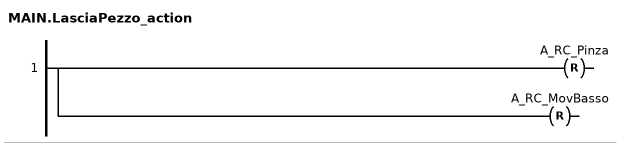
[picture p96: MAIN.LasciaPezzo_action (LD)]
_LD_ (* Ladder Diagram *)
NETWORK 1
	* --- (R A_RC_Pinza) (R A_RC_MovBasso)
_END_LD_
(* the same logic as Structured Text *)
(* Network 1 *)
A_RC_Pinza := FALSE;
A_RC_MovBasso := FALSE;
END_ACTION

ACTION PinzaSet21_action:
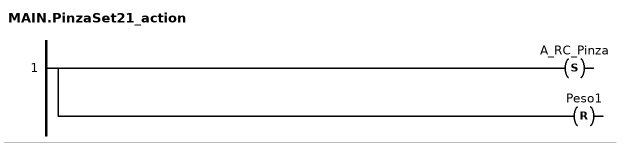
_LD_ (* Ladder Diagram *)
NETWORK 1
	* --- (S A_RC_Pinza) (R Peso1)
_END_LD_
(* the same logic as Structured Text *)
(* Network 1 *)
A_RC_Pinza := TRUE;
Peso1 := FALSE;
END_ACTION

ACTION MovA1_action:
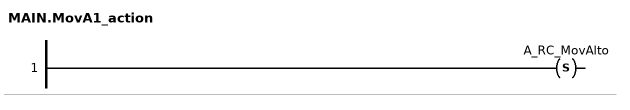
_LD_ (* Ladder Diagram *)
NETWORK 1
	* --- (S A_RC_MovAlto)
_END_LD_
(* the same logic as Structured Text *)
(* Network 1 *)
A_RC_MovAlto := TRUE;
END_ACTION

ACTION MovS1RA_action:
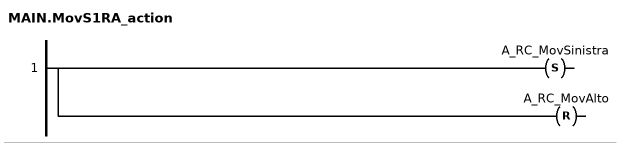
_LD_ (* Ladder Diagram *)
NETWORK 1
	* --- (S A_RC_MovSinistra) (R A_RC_MovAlto)
_END_LD_
(* the same logic as Structured Text *)
(* Network 1 *)
A_RC_MovSinistra := TRUE;
A_RC_MovAlto := FALSE;
END_ACTION

ACTION PinzaSet22_action:
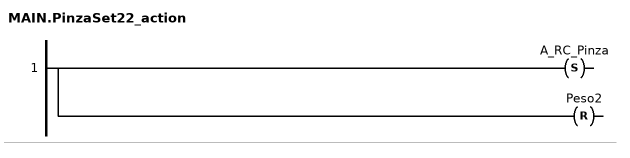
_LD_ (* Ladder Diagram *)
NETWORK 1
	* --- (S A_RC_Pinza) (R Peso2)
_END_LD_
(* the same logic as Structured Text *)
(* Network 1 *)
A_RC_Pinza := TRUE;
Peso2 := FALSE;
END_ACTION

ACTION MovA2_action:
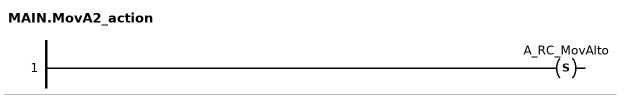
_LD_ (* Ladder Diagram *)
NETWORK 1
	* --- (S A_RC_MovAlto)
_END_LD_
(* the same logic as Structured Text *)
(* Network 1 *)
A_RC_MovAlto := TRUE;
END_ACTION

ACTION MovS2RA_action:
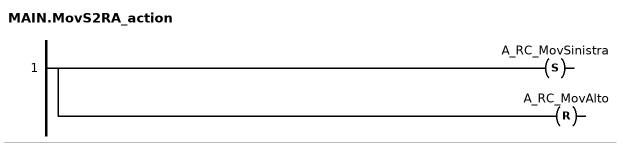
_LD_ (* Ladder Diagram *)
NETWORK 1
	* --- (S A_RC_MovSinistra) (R A_RC_MovAlto)
_END_LD_
(* the same logic as Structured Text *)
(* Network 1 *)
A_RC_MovSinistra := TRUE;
A_RC_MovAlto := FALSE;
END_ACTION

ACTION PinzaSet23_action:
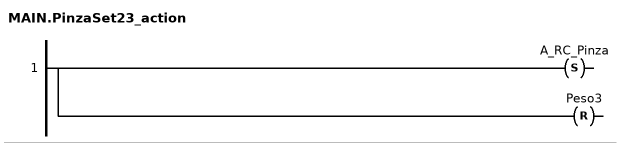
_LD_ (* Ladder Diagram *)
NETWORK 1
	* --- (S A_RC_Pinza) (R Peso3)
_END_LD_
(* the same logic as Structured Text *)
(* Network 1 *)
A_RC_Pinza := TRUE;
Peso3 := FALSE;
END_ACTION

ACTION MovA3_action:
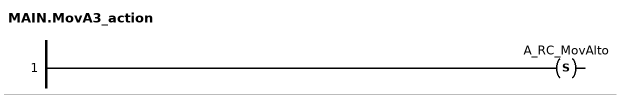
_LD_ (* Ladder Diagram *)
NETWORK 1
	* --- (S A_RC_MovAlto)
_END_LD_
(* the same logic as Structured Text *)
(* Network 1 *)
A_RC_MovAlto := TRUE;
END_ACTION

ACTION MovS3RA_action:
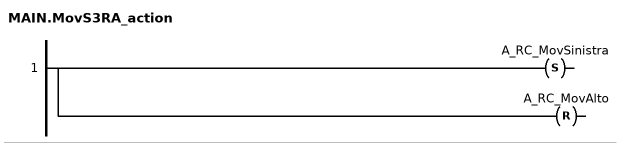
_LD_ (* Ladder Diagram *)
NETWORK 1
	* --- (S A_RC_MovSinistra) (R A_RC_MovAlto)
_END_LD_
(* the same logic as Structured Text *)
(* Network 1 *)
A_RC_MovSinistra := TRUE;
A_RC_MovAlto := FALSE;
END_ACTION

ACTION Stab_action:
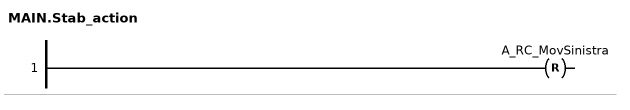
_LD_ (* Ladder Diagram *)
NETWORK 1
	* --- (R A_RC_MovSinistra)
_END_LD_
(* the same logic as Structured Text *)
(* Network 1 *)
A_RC_MovSinistra := FALSE;
END_ACTION

ACTION Release_action:
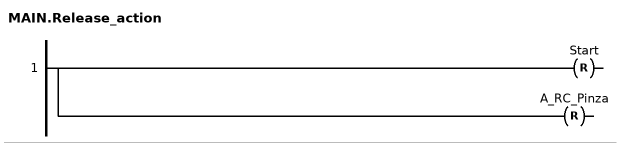
_LD_ (* Ladder Diagram *)
NETWORK 1
	* --- (R Start) (R A_RC_Pinza)
_END_LD_
(* the same logic as Structured Text *)
(* Network 1 *)
Start := FALSE;
A_RC_Pinza := FALSE;
END_ACTION

ACTION FermaUp_action:
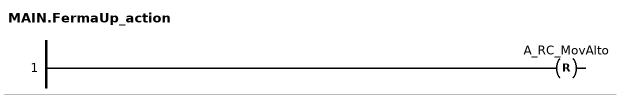
_LD_ (* Ladder Diagram *)
NETWORK 1
	* --- (R A_RC_MovAlto)
_END_LD_
(* the same logic as Structured Text *)
(* Network 1 *)
A_RC_MovAlto := FALSE;
END_ACTION

ACTION ResetEspelli_action:
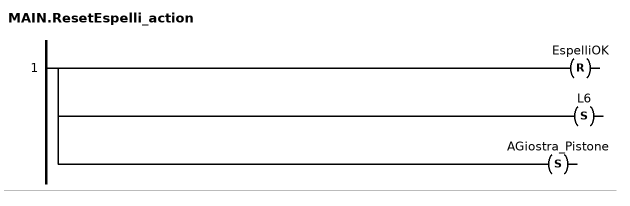
_LD_ (* Ladder Diagram *)
NETWORK 1
	* --- (R EspelliOK) (S L6) (S AGiostra_Pistone)
_END_LD_
(* the same logic as Structured Text *)
(* Network 1 *)
EspelliOK := FALSE;
L6 := TRUE;
AGiostra_Pistone := TRUE;
END_ACTION

ACTION ResetPistone_action:
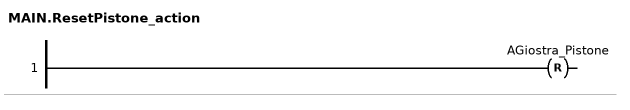
_LD_ (* Ladder Diagram *)
NETWORK 1
	* --- (R AGiostra_Pistone)
_END_LD_
(* the same logic as Structured Text *)
(* Network 1 *)
AGiostra_Pistone := FALSE;
END_ACTION

ACTION ResetL6_action:
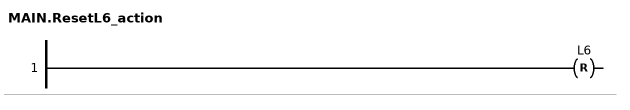
_LD_ (* Ladder Diagram *)
NETWORK 1
	* --- (R L6)
_END_LD_
(* the same logic as Structured Text *)
(* Network 1 *)
L6 := FALSE;
END_ACTION

ACTION Rot14_action:
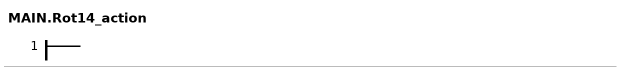
_LD_ (* Ladder Diagram *)
NETWORK 1
	*
_END_LD_
(* the same logic as Structured Text *)
(* Network 1 *)
END_ACTION

TRANSITION tra0:
_LD_ (* Ladder Diagram *)
NETWORK 1
	[SAsc_Capacitivo] - T32:TON(IN: *, PT: T#1000ms)
_END_LD_
(* the same logic as Structured Text *)
(* Network 1 *)
T32(IN := SAsc_Capacitivo, PT := T#1000ms);
tra0 := T32.Q;
END_TRANSITION

TRANSITION tra1:
_LD_ (* Ladder Diagram *)
NETWORK 1
	[SAsc_Alto] - [/SAsc_Altezza] - T33:TON(IN: *, PT: T#1000ms)
_END_LD_
(* the same logic as Structured Text *)
(* Network 1 *)
T33(IN := SAsc_Alto AND NOT SAsc_Altezza, PT := T#1000ms);
tra1 := T33.Q;
END_TRANSITION

TRANSITION trans4:
_LD_ (* Ladder Diagram *)
NETWORK 1
	[SAsc_Basso] - T35:TON(IN: *, PT: T#100ms)
_END_LD_
(* the same logic as Structured Text *)
(* Network 1 *)
T35(IN := SAsc_Basso, PT := T#100ms);
trans4 := T35.Q;
END_TRANSITION

TRANSITION trans6:
_LD_ (* Ladder Diagram *)
NETWORK 1
	[AAsc_pistone] - T39:TON(IN: *, PT: T#500ms)
_END_LD_
(* the same logic as Structured Text *)
(* Network 1 *)
T39(IN := AAsc_pistone, PT := T#500ms);
trans6 := T39.Q;
END_TRANSITION

TRANSITION trans14:
_LD_ (* Ladder Diagram *)
NETWORK 1
	[ARullo_pistone] - T36:TON(IN: *, PT: T#500ms)
_END_LD_
(* the same logic as Structured Text *)
(* Network 1 *)
T36(IN := ARullo_pistone, PT := T#500ms);
trans14 := T36.Q;
END_TRANSITION

TRANSITION tra2:
_LD_ (* Ladder Diagram *)
NETWORK 1
	[SAsc_Altezza] - [SAsc_Alto] - T34:TON(IN: *, PT: T#1000ms)
_END_LD_
(* the same logic as Structured Text *)
(* Network 1 *)
T34(IN := SAsc_Altezza AND SAsc_Alto, PT := T#1000ms);
tra2 := T34.Q;
END_TRANSITION

TRANSITION trans3:
_LD_ (* Ladder Diagram *)
NETWORK 1
	[AAsc_pistone] - T37:TON(IN: *, PT: T#500ms)
_END_LD_
(* the same logic as Structured Text *)
(* Network 1 *)
T37(IN := AAsc_pistone, PT := T#500ms);
trans3 := T37.Q;
END_TRANSITION

TRANSITION Transotto:
_LD_ (* Ladder Diagram *)
NETWORK 1
	[SAsc_Basso] - T38:TON(IN: *, PT: T#100ms)
_END_LD_
(* the same logic as Structured Text *)
(* Network 1 *)
T38(IN := SAsc_Basso, PT := T#100ms);
Transotto := T38.Q;
END_TRANSITION

TRANSITION Trans76:
_LD_ (* Ladder Diagram *)
NETWORK 1
	[/VarOFF] - T6:TON(IN: *, PT: T#500ms)
_END_LD_
(* the same logic as Structured Text *)
(* Network 1 *)
T6(IN := NOT VarOFF, PT := T#500ms);
Trans76 := T6.Q;
END_TRANSITION

TRANSITION tfftftft:
_LD_ (* Ladder Diagram *)
NETWORK 1
	[/VarON] - T7:TON(IN: *, PT: T#500ms)
_END_LD_
(* the same logic as Structured Text *)
(* Network 1 *)
T7(IN := NOT VarON, PT := T#500ms);
tfftftft := T7.Q;
END_TRANSITION

TRANSITION FineC:
_LD_ (* Ladder Diagram *)
NETWORK 1
	[/SRullo_Finecorsa] - T3:TON(IN: *, PT: T#100ms)
_END_LD_
(* the same logic as Structured Text *)
(* Network 1 *)
T3(IN := NOT SRullo_Finecorsa, PT := T#100ms);
FineC := T3.Q;
END_TRANSITION

TRANSITION Trans16:
_LD_ (* Ladder Diagram *)
NETWORK 1 (ci sono pezzi):
	[RulloVuoto] - [L0] - T4:TON(IN: *, PT: T#1400ms)
_END_LD_
(* the same logic as Structured Text *)
(* Network 1 *)
(* label: (ci sono pezzi) *)
T4(IN := RulloVuoto AND L0, PT := T#1400ms);
Trans16 := T4.Q;
END_TRANSITION

TRANSITION Check+G:
_LD_ (* Ladder Diagram *)
NETWORK 1
	[/L0] - [/L1] - [/L2] - [/L3] - [/L4] - [/L5] - [/L6] - [/GiostraOK] - [/Tempo]
_END_LD_
(* the same logic as Structured Text *)
(* Network 1 *)
Check_G := NOT L0 AND NOT L1 AND NOT L2 AND NOT L3 AND NOT L4 AND NOT L5 AND NOT L6 AND NOT GiostraOK AND NOT Tempo;
END_TRANSITION

TRANSITION Trans71:
_LD_ (* Ladder Diagram *)
NETWORK 1 (non ci sono piu pezzi sul nastro):
	[/RulloVuoto] - [L0] - T5:TON(IN: *, PT: T#1400ms)
_END_LD_
(* the same logic as Structured Text *)
(* Network 1 *)
(* label: (non ci sono piu pezzi sul nastro) *)
T5(IN := NOT RulloVuoto AND L0, PT := T#1400ms);
Trans71 := T5.Q;
END_TRANSITION

TRANSITION Check+G:
_LD_ (* Ladder Diagram *)
NETWORK 1
	[/L0] - [/L1] - [/L2] - [/L3] - [/L4] - [/L5] - [/L6] - [/GiostraOK] - [/Tempo]
_END_LD_
(* the same logic as Structured Text *)
(* Network 1 *)
Check_G := NOT L0 AND NOT L1 AND NOT L2 AND NOT L3 AND NOT L4 AND NOT L5 AND NOT L6 AND NOT GiostraOK AND NOT Tempo;
END_TRANSITION

TRANSITION Check+T:
_LD_ (* Ladder Diagram *)
NETWORK 1
	[/L0] - [/L1] - [/L2] - [/L3] - [/L4] - [/L5] - [/L6] - [/Tempo]
_END_LD_
(* the same logic as Structured Text *)
(* Network 1 *)
Check_T := NOT L0 AND NOT L1 AND NOT L2 AND NOT L3 AND NOT L4 AND NOT L5 AND NOT L6 AND NOT Tempo;
END_TRANSITION

TRANSITION Check+T:
_LD_ (* Ladder Diagram *)
NETWORK 1
	[/L0] - [/L1] - [/L2] - [/L3] - [/L4] - [/L5] - [/L6] - [/Tempo]
_END_LD_
(* the same logic as Structured Text *)
(* Network 1 *)
Check_T := NOT L0 AND NOT L1 AND NOT L2 AND NOT L3 AND NOT L4 AND NOT L5 AND NOT L6 AND NOT Tempo;
END_TRANSITION

TRANSITION Trans20:
_LD_ (* Ladder Diagram *)
NETWORK 1
	[AGiostra_Gira] - T8:TON(IN: *, PT: T#1300ms)
_END_LD_
(* the same logic as Structured Text *)
(* Network 1 *)
T8(IN := AGiostra_Gira, PT := T#1300ms);
Trans20 := T8.Q;
END_TRANSITION

TRANSITION Check:
_LD_ (* Ladder Diagram *)
NETWORK 1
	[/L0] - [/L1] - [/L2] - [/L3] - [/L4] - [/L5] - [/L6]
_END_LD_
(* the same logic as Structured Text *)
(* Network 1 *)
Check := NOT L0 AND NOT L1 AND NOT L2 AND NOT L3 AND NOT L4 AND NOT L5 AND NOT L6;
END_TRANSITION

TRANSITION TColore:
_LD_ (* Ladder Diagram *)
NETWORK 1
	[ColoreOK] - [/Tempo]
_END_LD_
(* the same logic as Structured Text *)
(* Network 1 *)
TColore := ColoreOK AND NOT Tempo;
END_TRANSITION

TRANSITION Rosso:
_LD_ (* Ladder Diagram *)
NETWORK 1
	[SGiostra_Colore] - [/AGiostra_Gira] - T9:TON(IN: *, PT: T#500ms)
_END_LD_
(* the same logic as Structured Text *)
(* Network 1 *)
T9(IN := SGiostra_Colore AND NOT AGiostra_Gira, PT := T#500ms);
Rosso := T9.Q;
END_TRANSITION

TRANSITION Check+G:
_LD_ (* Ladder Diagram *)
NETWORK 1
	[/L0] - [/L1] - [/L2] - [/L3] - [/L4] - [/L5] - [/L6] - [/GiostraOK] - [/Tempo]
_END_LD_
(* the same logic as Structured Text *)
(* Network 1 *)
Check_G := NOT L0 AND NOT L1 AND NOT L2 AND NOT L3 AND NOT L4 AND NOT L5 AND NOT L6 AND NOT GiostraOK AND NOT Tempo;
END_TRANSITION

TRANSITION Check+T:
_LD_ (* Ladder Diagram *)
NETWORK 1
	[/L0] - [/L1] - [/L2] - [/L3] - [/L4] - [/L5] - [/L6] - [/Tempo]
_END_LD_
(* the same logic as Structured Text *)
(* Network 1 *)
Check_T := NOT L0 AND NOT L1 AND NOT L2 AND NOT L3 AND NOT L4 AND NOT L5 AND NOT L6 AND NOT Tempo;
END_TRANSITION

TRANSITION NonRosso:
_LD_ (* Ladder Diagram *)
NETWORK 1
	[/SGiostra_Colore] - [/AGiostra_Gira] - T10:TON(IN: *, PT: T#500ms)
_END_LD_
(* the same logic as Structured Text *)
(* Network 1 *)
T10(IN := NOT SGiostra_Colore AND NOT AGiostra_Gira, PT := T#500ms);
NonRosso := T10.Q;
END_TRANSITION

TRANSITION Check+G:
_LD_ (* Ladder Diagram *)
NETWORK 1
	[/L0] - [/L1] - [/L2] - [/L3] - [/L4] - [/L5] - [/L6] - [/GiostraOK] - [/Tempo]
_END_LD_
(* the same logic as Structured Text *)
(* Network 1 *)
Check_G := NOT L0 AND NOT L1 AND NOT L2 AND NOT L3 AND NOT L4 AND NOT L5 AND NOT L6 AND NOT GiostraOK AND NOT Tempo;
END_TRANSITION

TRANSITION Check+T:
_LD_ (* Ladder Diagram *)
NETWORK 1
	[/L0] - [/L1] - [/L2] - [/L3] - [/L4] - [/L5] - [/L6] - [/Tempo]
_END_LD_
(* the same logic as Structured Text *)
(* Network 1 *)
Check_T := NOT L0 AND NOT L1 AND NOT L2 AND NOT L3 AND NOT L4 AND NOT L5 AND NOT L6 AND NOT Tempo;
END_TRANSITION

TRANSITION TTrapano:
_LD_ (* Ladder Diagram *)
NETWORK 1
	[TrapanoOK] - [/Tempo]
_END_LD_
(* the same logic as Structured Text *)
(* Network 1 *)
TTrapano := TrapanoOK AND NOT Tempo;
END_TRANSITION

TRANSITION Bucare:
_LD_ (* Ladder Diagram *)
NETWORK 1
	[P2C1B0] - [SDremel_alto]
_END_LD_
(* the same logic as Structured Text *)
(* Network 1 *)
Bucare := P2C1B0 AND SDremel_alto;
END_TRANSITION

TRANSITION SDremel_Basso:
_LD_ (* Ladder Diagram *)
NETWORK 1
	[SDremel_Basso] - T11:TON(IN: *, PT: T#1000ms)
_END_LD_
(* the same logic as Structured Text *)
(* Network 1 *)
T11(IN := SDremel_Basso, PT := T#1000ms);
SDremel_Basso := T11.Q;
END_TRANSITION

TRANSITION Check+G:
_LD_ (* Ladder Diagram *)
NETWORK 1
	[/L0] - [/L1] - [/L2] - [/L3] - [/L4] - [/L5] - [/L6] - [/GiostraOK] - [/Tempo]
_END_LD_
(* the same logic as Structured Text *)
(* Network 1 *)
Check_G := NOT L0 AND NOT L1 AND NOT L2 AND NOT L3 AND NOT L4 AND NOT L5 AND NOT L6 AND NOT GiostraOK AND NOT Tempo;
END_TRANSITION

TRANSITION Check+T:
_LD_ (* Ladder Diagram *)
NETWORK 1
	[/L0] - [/L1] - [/L2] - [/L3] - [/L4] - [/L5] - [/L6] - [/Tempo]
_END_LD_
(* the same logic as Structured Text *)
(* Network 1 *)
Check_T := NOT L0 AND NOT L1 AND NOT L2 AND NOT L3 AND NOT L4 AND NOT L5 AND NOT L6 AND NOT Tempo;
END_TRANSITION

TRANSITION NonBucare:
_LD_ (* Ladder Diagram *)
NETWORK 1
	[P2C0B0] - [/AGiostra_Gira]
_END_LD_
(* the same logic as Structured Text *)
(* Network 1 *)
NonBucare := P2C0B0 AND NOT AGiostra_Gira;
END_TRANSITION

TRANSITION Check+G:
_LD_ (* Ladder Diagram *)
NETWORK 1
	[/L0] - [/L1] - [/L2] - [/L3] - [/L4] - [/L5] - [/L6] - [/GiostraOK] - [/Tempo]
_END_LD_
(* the same logic as Structured Text *)
(* Network 1 *)
Check_G := NOT L0 AND NOT L1 AND NOT L2 AND NOT L3 AND NOT L4 AND NOT L5 AND NOT L6 AND NOT GiostraOK AND NOT Tempo;
END_TRANSITION

TRANSITION Check+T:
_LD_ (* Ladder Diagram *)
NETWORK 1
	[/L0] - [/L1] - [/L2] - [/L3] - [/L4] - [/L5] - [/L6] - [/Tempo]
_END_LD_
(* the same logic as Structured Text *)
(* Network 1 *)
Check_T := NOT L0 AND NOT L1 AND NOT L2 AND NOT L3 AND NOT L4 AND NOT L5 AND NOT L6 AND NOT Tempo;
END_TRANSITION

TRANSITION TTastatore:
_LD_ (* Ladder Diagram *)
NETWORK 1
	[TastatoreOK] - [/Tempo]
_END_LD_
(* the same logic as Structured Text *)
(* Network 1 *)
TTastatore := TastatoreOK AND NOT Tempo;
END_TRANSITION

TRANSITION Tast1:
_LD_ (* Ladder Diagram *)
NETWORK 1
	[P3C1B1] - [/AGiostra_Gira]
_END_LD_
(* the same logic as Structured Text *)
(* Network 1 *)
Tast1 := P3C1B1 AND NOT AGiostra_Gira;
END_TRANSITION

TRANSITION Bucato:
_LD_ (* Ladder Diagram *)
NETWORK 1
	[AGiostra_Altezza] - [SGiostra_Altezza] - T12:TON(IN: *, PT: T#1500ms)
_END_LD_
(* the same logic as Structured Text *)
(* Network 1 *)
T12(IN := AGiostra_Altezza AND SGiostra_Altezza, PT := T#1500ms);
Bucato := T12.Q;
END_TRANSITION

TRANSITION Check+G:
_LD_ (* Ladder Diagram *)
NETWORK 1
	[/L0] - [/L1] - [/L2] - [/L3] - [/L4] - [/L5] - [/L6] - [/GiostraOK] - [/Tempo]
_END_LD_
(* the same logic as Structured Text *)
(* Network 1 *)
Check_G := NOT L0 AND NOT L1 AND NOT L2 AND NOT L3 AND NOT L4 AND NOT L5 AND NOT L6 AND NOT GiostraOK AND NOT Tempo;
END_TRANSITION

TRANSITION Check+T:
_LD_ (* Ladder Diagram *)
NETWORK 1
	[/L0] - [/L1] - [/L2] - [/L3] - [/L4] - [/L5] - [/L6] - [/Tempo]
_END_LD_
(* the same logic as Structured Text *)
(* Network 1 *)
Check_T := NOT L0 AND NOT L1 AND NOT L2 AND NOT L3 AND NOT L4 AND NOT L5 AND NOT L6 AND NOT Tempo;
END_TRANSITION

TRANSITION NonBucato:
_LD_ (* Ladder Diagram *)
NETWORK 1
	[/SGiostra_Altezza] - [AGiostra_Altezza] - T13:TON(IN: *, PT: T#1500ms)
_END_LD_
(* the same logic as Structured Text *)
(* Network 1 *)
T13(IN := NOT SGiostra_Altezza AND AGiostra_Altezza, PT := T#1500ms);
NonBucato := T13.Q;
END_TRANSITION

TRANSITION Check+G:
_LD_ (* Ladder Diagram *)
NETWORK 1
	[/L0] - [/L1] - [/L2] - [/L3] - [/L4] - [/L5] - [/L6] - [/GiostraOK] - [/Tempo]
_END_LD_
(* the same logic as Structured Text *)
(* Network 1 *)
Check_G := NOT L0 AND NOT L1 AND NOT L2 AND NOT L3 AND NOT L4 AND NOT L5 AND NOT L6 AND NOT GiostraOK AND NOT Tempo;
END_TRANSITION

TRANSITION Check+T:
_LD_ (* Ladder Diagram *)
NETWORK 1
	[/L0] - [/L1] - [/L2] - [/L3] - [/L4] - [/L5] - [/L6] - [/Tempo]
_END_LD_
(* the same logic as Structured Text *)
(* Network 1 *)
Check_T := NOT L0 AND NOT L1 AND NOT L2 AND NOT L3 AND NOT L4 AND NOT L5 AND NOT L6 AND NOT Tempo;
END_TRANSITION

TRANSITION Tast2:
_LD_ (* Ladder Diagram *)
NETWORK 1
	[P3C0B0] - [/AGiostra_Gira]
_END_LD_
(* the same logic as Structured Text *)
(* Network 1 *)
Tast2 := P3C0B0 AND NOT AGiostra_Gira;
END_TRANSITION

TRANSITION Check+G:
_LD_ (* Ladder Diagram *)
NETWORK 1
	[/L0] - [/L1] - [/L2] - [/L3] - [/L4] - [/L5] - [/L6] - [/GiostraOK] - [/Tempo]
_END_LD_
(* the same logic as Structured Text *)
(* Network 1 *)
Check_G := NOT L0 AND NOT L1 AND NOT L2 AND NOT L3 AND NOT L4 AND NOT L5 AND NOT L6 AND NOT GiostraOK AND NOT Tempo;
END_TRANSITION

TRANSITION Check+T:
_LD_ (* Ladder Diagram *)
NETWORK 1
	[/L0] - [/L1] - [/L2] - [/L3] - [/L4] - [/L5] - [/L6] - [/Tempo]
_END_LD_
(* the same logic as Structured Text *)
(* Network 1 *)
Check_T := NOT L0 AND NOT L1 AND NOT L2 AND NOT L3 AND NOT L4 AND NOT L5 AND NOT L6 AND NOT Tempo;
END_TRANSITION

TRANSITION TMarker:
_LD_ (* Ladder Diagram *)
NETWORK 1
	[/Tempo] - [MarkerOK]
_END_LD_
(* the same logic as Structured Text *)
(* Network 1 *)
TMarker := NOT Tempo AND MarkerOK;
END_TRANSITION

TRANSITION Colora:
_LD_ (* Ladder Diagram *)
NETWORK 1
	[P4C0B0] - [/AGiostra_Gira]
_END_LD_
(* the same logic as Structured Text *)
(* Network 1 *)
Colora := P4C0B0 AND NOT AGiostra_Gira;
END_TRANSITION

TRANSITION NonColora:
_LD_ (* Ladder Diagram *)
NETWORK 1
	[NC] - [/AGiostra_Gira]
_END_LD_
(* the same logic as Structured Text *)
(* Network 1 *)
NonColora := NC AND NOT AGiostra_Gira;
END_TRANSITION

TRANSITION NonColoraW:
_LD_ (* Ladder Diagram *)
NETWORK 1
	[P4C1B1W] - [SGiostra_MarkerAlto]
_END_LD_
(* the same logic as Structured Text *)
(* Network 1 *)
NonColoraW := P4C1B1W AND SGiostra_MarkerAlto;
END_TRANSITION

TRANSITION NonColoraR:
_LD_ (* Ladder Diagram *)
NETWORK 1
	[P4C1B1R] - [SGiostra_MarkerAlto]
_END_LD_
(* the same logic as Structured Text *)
(* Network 1 *)
NonColoraR := P4C1B1R AND SGiostra_MarkerAlto;
END_TRANSITION

TRANSITION Check+G:
_LD_ (* Ladder Diagram *)
NETWORK 1
	[/L0] - [/L1] - [/L2] - [/L3] - [/L4] - [/L5] - [/L6] - [/GiostraOK] - [/Tempo]
_END_LD_
(* the same logic as Structured Text *)
(* Network 1 *)
Check_G := NOT L0 AND NOT L1 AND NOT L2 AND NOT L3 AND NOT L4 AND NOT L5 AND NOT L6 AND NOT GiostraOK AND NOT Tempo;
END_TRANSITION

TRANSITION Check+T:
_LD_ (* Ladder Diagram *)
NETWORK 1
	[/L0] - [/L1] - [/L2] - [/L3] - [/L4] - [/L5] - [/L6] - [/Tempo]
_END_LD_
(* the same logic as Structured Text *)
(* Network 1 *)
Check_T := NOT L0 AND NOT L1 AND NOT L2 AND NOT L3 AND NOT L4 AND NOT L5 AND NOT L6 AND NOT Tempo;
END_TRANSITION

TRANSITION Check+G:
_LD_ (* Ladder Diagram *)
NETWORK 1
	[/L0] - [/L1] - [/L2] - [/L3] - [/L4] - [/L5] - [/L6] - [/GiostraOK] - [/Tempo]
_END_LD_
(* the same logic as Structured Text *)
(* Network 1 *)
Check_G := NOT L0 AND NOT L1 AND NOT L2 AND NOT L3 AND NOT L4 AND NOT L5 AND NOT L6 AND NOT GiostraOK AND NOT Tempo;
END_TRANSITION

TRANSITION Check+T:
_LD_ (* Ladder Diagram *)
NETWORK 1
	[/L0] - [/L1] - [/L2] - [/L3] - [/L4] - [/L5] - [/L6] - [/Tempo]
_END_LD_
(* the same logic as Structured Text *)
(* Network 1 *)
Check_T := NOT L0 AND NOT L1 AND NOT L2 AND NOT L3 AND NOT L4 AND NOT L5 AND NOT L6 AND NOT Tempo;
END_TRANSITION

TRANSITION Trans54:
_LD_ (* Ladder Diagram *)
NETWORK 1
	[SGiostra_MarkerBasso] - T14:TON(IN: *, PT: T#600ms)
_END_LD_
(* the same logic as Structured Text *)
(* Network 1 *)
T14(IN := SGiostra_MarkerBasso, PT := T#600ms);
Trans54 := T14.Q;
END_TRANSITION

TRANSITION Trans80:
_LD_ (* Ladder Diagram *)
NETWORK 1
	[/AGiostra_Marker] - T15:TON(IN: *, PT: T#800ms)
_END_LD_
(* the same logic as Structured Text *)
(* Network 1 *)
T15(IN := NOT AGiostra_Marker, PT := T#800ms);
Trans80 := T15.Q;
END_TRANSITION

TRANSITION Check+G:
_LD_ (* Ladder Diagram *)
NETWORK 1
	[/L0] - [/L1] - [/L2] - [/L3] - [/L4] - [/L5] - [/L6] - [/GiostraOK] - [/Tempo]
_END_LD_
(* the same logic as Structured Text *)
(* Network 1 *)
Check_G := NOT L0 AND NOT L1 AND NOT L2 AND NOT L3 AND NOT L4 AND NOT L5 AND NOT L6 AND NOT GiostraOK AND NOT Tempo;
END_TRANSITION

TRANSITION Check+T:
_LD_ (* Ladder Diagram *)
NETWORK 1
	[/L0] - [/L1] - [/L2] - [/L3] - [/L4] - [/L5] - [/L6] - [/Tempo]
_END_LD_
(* the same logic as Structured Text *)
(* Network 1 *)
Check_T := NOT L0 AND NOT L1 AND NOT L2 AND NOT L3 AND NOT L4 AND NOT L5 AND NOT L6 AND NOT Tempo;
END_TRANSITION

TRANSITION TScarto:
_LD_ (* Ladder Diagram *)
NETWORK 1
	[ScartoOK] - [/Tempo]
_END_LD_
(* the same logic as Structured Text *)
(* Network 1 *)
TScarto := ScartoOK AND NOT Tempo;
END_TRANSITION

TRANSITION Scartare:
_LD_ (* Ladder Diagram *)
NETWORK 1
	[P5C1B1W] - T20:TON(IN: *, PT: T#200ms)
_END_LD_
(* the same logic as Structured Text *)
(* Network 1 *)
T20(IN := P5C1B1W, PT := T#200ms);
Scartare := T20.Q;
END_TRANSITION

TRANSITION Trans67:
_LD_ (* Ladder Diagram *)
NETWORK 1
	[AGiostra_Scarta] - T16:TON(IN: *, PT: T#1000ms)
_END_LD_
(* the same logic as Structured Text *)
(* Network 1 *)
T16(IN := AGiostra_Scarta, PT := T#1000ms);
Trans67 := T16.Q;
END_TRANSITION

TRANSITION AttesaIndietro:
_LD_ (* Ladder Diagram *)
NETWORK 1
	[/AGiostra_Scarta] - T17:TON(IN: *, PT: T#500ms)
_END_LD_
(* the same logic as Structured Text *)
(* Network 1 *)
T17(IN := NOT AGiostra_Scarta, PT := T#500ms);
AttesaIndietro := T17.Q;
END_TRANSITION

TRANSITION Check+G:
_LD_ (* Ladder Diagram *)
NETWORK 1
	[/L0] - [/L1] - [/L2] - [/L3] - [/L4] - [/L5] - [/L6] - [/GiostraOK] - [/Tempo]
_END_LD_
(* the same logic as Structured Text *)
(* Network 1 *)
Check_G := NOT L0 AND NOT L1 AND NOT L2 AND NOT L3 AND NOT L4 AND NOT L5 AND NOT L6 AND NOT GiostraOK AND NOT Tempo;
END_TRANSITION

TRANSITION Nonscartare:
_LD_ (* Ladder Diagram *)
NETWORK 1
	{ [P5C1B1R] | [P5C0B0] } - T22:TON(IN: *, PT: T#500ms)
_END_LD_
(* the same logic as Structured Text *)
(* Network 1 *)
T22(IN := P5C1B1R OR P5C0B0, PT := T#500ms);
Nonscartare := T22.Q;
END_TRANSITION

TRANSITION Check+G:
_LD_ (* Ladder Diagram *)
NETWORK 1
	[/L0] - [/L1] - [/L2] - [/L3] - [/L4] - [/L5] - [/L6] - [/GiostraOK] - [/Tempo]
_END_LD_
(* the same logic as Structured Text *)
(* Network 1 *)
Check_G := NOT L0 AND NOT L1 AND NOT L2 AND NOT L3 AND NOT L4 AND NOT L5 AND NOT L6 AND NOT GiostraOK AND NOT Tempo;
END_TRANSITION

TRANSITION Check+T:
_LD_ (* Ladder Diagram *)
NETWORK 1
	[/L0] - [/L1] - [/L2] - [/L3] - [/L4] - [/L5] - [/L6] - [/Tempo]
_END_LD_
(* the same logic as Structured Text *)
(* Network 1 *)
Check_T := NOT L0 AND NOT L1 AND NOT L2 AND NOT L3 AND NOT L4 AND NOT L5 AND NOT L6 AND NOT Tempo;
END_TRANSITION

TRANSITION ControlloFCSX:
_LD_ (* Ladder Diagram *)
NETWORK 1
	[S_RC_FineCorsaSinistra]
_END_LD_
(* the same logic as Structured Text *)
(* Network 1 *)
ControlloFCSX := S_RC_FineCorsaSinistra;
END_TRANSITION

TRANSITION ControlloFCDX:
_LD_ (* Ladder Diagram *)
NETWORK 1
	[/S_RC_FineCorsaDestra]
_END_LD_
(* the same logic as Structured Text *)
(* Network 1 *)
ControlloFCDX := NOT S_RC_FineCorsaDestra;
END_TRANSITION

TRANSITION SbloccoDx:
_LD_ (* Ladder Diagram *)
NETWORK 1
	[S_RC_FineCorsaDestra]
_END_LD_
(* the same logic as Structured Text *)
(* Network 1 *)
SbloccoDx := S_RC_FineCorsaDestra;
END_TRANSITION

TRANSITION ControlloFCDown:
_LD_ (* Ladder Diagram *)
NETWORK 1
	[/S_RC_FineCorsaBasso]
_END_LD_
(* the same logic as Structured Text *)
(* Network 1 *)
ControlloFCDown := NOT S_RC_FineCorsaBasso;
END_TRANSITION

TRANSITION SbloccoDown:
_LD_ (* Ladder Diagram *)
NETWORK 1
	[S_RC_FineCorsaBasso]
_END_LD_
(* the same logic as Structured Text *)
(* Network 1 *)
SbloccoDown := S_RC_FineCorsaBasso;
END_TRANSITION

TRANSITION CheckStart:
_LD_ (* Ladder Diagram *)
NETWORK 1
	[/Start]
_END_LD_
(* the same logic as Structured Text *)
(* Network 1 *)
CheckStart := NOT Start;
END_TRANSITION

TRANSITION Salita:
_LD_ (* Ladder Diagram *)
NETWORK 1
	[StopSali]
_END_LD_
(* the same logic as Structured Text *)
(* Network 1 *)
Salita := StopSali;
END_TRANSITION

TRANSITION Bea:
_LD_ (* Ladder Diagram *)
NETWORK 1
	[/A_RC_MovAlto] - [/A_RC_MovBasso]
_END_LD_
(* the same logic as Structured Text *)
(* Network 1 *)
Bea := NOT A_RC_MovAlto AND NOT A_RC_MovBasso;
END_TRANSITION

TRANSITION Discesa:
_LD_ (* Ladder Diagram *)
NETWORK 1
	[StopScendi]
_END_LD_
(* the same logic as Structured Text *)
(* Network 1 *)
Discesa := StopScendi;
END_TRANSITION

TRANSITION Bea:
_LD_ (* Ladder Diagram *)
NETWORK 1
	[/A_RC_MovAlto] - [/A_RC_MovBasso]
_END_LD_
(* the same logic as Structured Text *)
(* Network 1 *)
Bea := NOT A_RC_MovAlto AND NOT A_RC_MovBasso;
END_TRANSITION

TRANSITION CheckStart1:
_LD_ (* Ladder Diagram *)
NETWORK 1
	[Start1]
_END_LD_
(* the same logic as Structured Text *)
(* Network 1 *)
CheckStart1 := Start1;
END_TRANSITION

TRANSITION FCSX:
_LD_ (* Ladder Diagram *)
NETWORK 1
	[S_RC_FineCorsaSinistra]
_END_LD_
(* the same logic as Structured Text *)
(* Network 1 *)
FCSX := S_RC_FineCorsaSinistra;
END_TRANSITION

TRANSITION ControlloStop:
_LD_ (* Ladder Diagram *)
NETWORK 1
	[/A_RC_MovDestra]
_END_LD_
(* the same logic as Structured Text *)
(* Network 1 *)
ControlloStop := NOT A_RC_MovDestra;
END_TRANSITION

TRANSITION Trans142:
_LD_ (* Ladder Diagram *)
NETWORK 1
	[/S_RC_ScivoloPieno] - T49:TON(IN: *, PT: T#1000ms)
_END_LD_
(* the same logic as Structured Text *)
(* Network 1 *)
T49(IN := NOT S_RC_ScivoloPieno, PT := T#1000ms);
Trans142 := T49.Q;
END_TRANSITION

TRANSITION trans143:
_LD_ (* Ladder Diagram *)
NETWORK 1
	[S_RC_ScivoloPieno] - T50:TON(IN: *, PT: T#1000ms)
_END_LD_
(* the same logic as Structured Text *)
(* Network 1 *)
T50(IN := S_RC_ScivoloPieno, PT := T#1000ms);
trans143 := T50.Q;
END_TRANSITION

TRANSITION RCCheck:
_LD_ (* Ladder Diagram *)
NETWORK 1
	[RAB] - [RSD] - [SGiostra_Presenza] - [/ScivoloPieno] - [/L6] - T40:TON(IN: *, PT: T#4000ms)
_END_LD_
(* the same logic as Structured Text *)
(* Network 1 *)
T40(IN := RAB AND RSD AND SGiostra_Presenza AND NOT ScivoloPieno AND NOT L6, PT := T#4000ms);
RCCheck := T40.Q;
END_TRANSITION

TRANSITION ABase:
_LD_ (* Ladder Diagram *)
NETWORK 1
	[AltBase]
_END_LD_
(* the same logic as Structured Text *)
(* Network 1 *)
ABase := AltBase;
END_TRANSITION

TRANSITION GripWait:
_LD_ (* Ladder Diagram *)
NETWORK 1
	[/A_RC_MovBasso] - T33:TON(IN: *, PT: T#500ms)
_END_LD_
(* the same logic as Structured Text *)
(* Network 1 *)
T33(IN := NOT A_RC_MovBasso, PT := T#500ms);
GripWait := T33.Q;
END_TRANSITION

TRANSITION CheckGrip:
_LD_ (* Ladder Diagram *)
NETWORK 1
	[A_RC_Pinza] - [/S_RC_PinzaSensore] - T34:TON(IN: *, PT: T#1000ms)
_END_LD_
(* the same logic as Structured Text *)
(* Network 1 *)
T34(IN := A_RC_Pinza AND NOT S_RC_PinzaSensore, PT := T#1000ms);
CheckGrip := T34.Q;
END_TRANSITION

TRANSITION AFinale:
_LD_ (* Ladder Diagram *)
NETWORK 1
	[AltFinale]
_END_LD_
(* the same logic as Structured Text *)
(* Network 1 *)
AFinale := AltFinale;
END_TRANSITION

TRANSITION LBilancia:
_LD_ (* Ladder Diagram *)
NETWORK 1 metti anche fine corsa per sicurezza:
	[Bilancia]
_END_LD_
(* the same logic as Structured Text *)
(* Network 1 *)
(* label: metti anche fine corsa per sicurezza *)
LBilancia := Bilancia;
END_TRANSITION

TRANSITION ABilancia:
_LD_ (* Ladder Diagram *)
NETWORK 1
	[AltBilancia]
_END_LD_
(* the same logic as Structured Text *)
(* Network 1 *)
ABilancia := AltBilancia;
END_TRANSITION

TRANSITION Peso1:
_LD_ (* Ladder Diagram *)
NETWORK 1
	[Peso1]
_END_LD_
(* the same logic as Structured Text *)
(* Network 1 *)
Peso1 := Peso1;
END_TRANSITION

TRANSITION CheckGrip1:
_LD_ (* Ladder Diagram *)
NETWORK 1
	[A_RC_Pinza] - [/S_RC_PinzaSensore] - T35:TON(IN: *, PT: T#1000ms)
_END_LD_
(* the same logic as Structured Text *)
(* Network 1 *)
T35(IN := A_RC_Pinza AND NOT S_RC_PinzaSensore, PT := T#1000ms);
CheckGrip1 := T35.Q;
END_TRANSITION

TRANSITION AScivolo:
_LD_ (* Ladder Diagram *)
NETWORK 1
	[AltScivolo]
_END_LD_
(* the same logic as Structured Text *)
(* Network 1 *)
AScivolo := AltScivolo;
END_TRANSITION

TRANSITION Scivolo1:
_LD_ (* Ladder Diagram *)
NETWORK 1
	[Scivolo1]
_END_LD_
(* the same logic as Structured Text *)
(* Network 1 *)
Scivolo1 := Scivolo1;
END_TRANSITION

TRANSITION Peso2:
_LD_ (* Ladder Diagram *)
NETWORK 1
	[Peso2]
_END_LD_
(* the same logic as Structured Text *)
(* Network 1 *)
Peso2 := Peso2;
END_TRANSITION

TRANSITION CheckGrip1:
_LD_ (* Ladder Diagram *)
NETWORK 1
	[A_RC_Pinza] - [/S_RC_PinzaSensore] - T36:TON(IN: *, PT: T#1000ms)
_END_LD_
(* the same logic as Structured Text *)
(* Network 1 *)
T36(IN := A_RC_Pinza AND NOT S_RC_PinzaSensore, PT := T#1000ms);
CheckGrip1 := T36.Q;
END_TRANSITION

TRANSITION AScivolo:
_LD_ (* Ladder Diagram *)
NETWORK 1
	[AltScivolo]
_END_LD_
(* the same logic as Structured Text *)
(* Network 1 *)
AScivolo := AltScivolo;
END_TRANSITION

TRANSITION Scivolo2:
_LD_ (* Ladder Diagram *)
NETWORK 1
	[Scivolo2]
_END_LD_
(* the same logic as Structured Text *)
(* Network 1 *)
Scivolo2 := Scivolo2;
END_TRANSITION

TRANSITION Peso3:
_LD_ (* Ladder Diagram *)
NETWORK 1
	[Peso3]
_END_LD_
(* the same logic as Structured Text *)
(* Network 1 *)
Peso3 := Peso3;
END_TRANSITION

TRANSITION CheckGrip1:
_LD_ (* Ladder Diagram *)
NETWORK 1
	[A_RC_Pinza] - [/S_RC_PinzaSensore] - T37:TON(IN: *, PT: T#1000ms)
_END_LD_
(* the same logic as Structured Text *)
(* Network 1 *)
T37(IN := A_RC_Pinza AND NOT S_RC_PinzaSensore, PT := T#1000ms);
CheckGrip1 := T37.Q;
END_TRANSITION

TRANSITION AScivolo:
_LD_ (* Ladder Diagram *)
NETWORK 1
	[AltScivolo]
_END_LD_
(* the same logic as Structured Text *)
(* Network 1 *)
AScivolo := AltScivolo;
END_TRANSITION

TRANSITION Scivolo3:
_LD_ (* Ladder Diagram *)
NETWORK 1
	[Scivolo3]
_END_LD_
(* the same logic as Structured Text *)
(* Network 1 *)
Scivolo3 := Scivolo3;
END_TRANSITION

TRANSITION WaitStab:
_LD_ (* Ladder Diagram *)
NETWORK 1
	[/A_RC_MovSinistra] - T38:TON(IN: *, PT: T#600ms)
_END_LD_
(* the same logic as Structured Text *)
(* Network 1 *)
T38(IN := NOT A_RC_MovSinistra, PT := T#600ms);
WaitStab := T38.Q;
END_TRANSITION

TRANSITION ControlloFCUP:
_LD_ (* Ladder Diagram *)
NETWORK 1
	[/S_RC_FineCorsaAlto]
_END_LD_
(* the same logic as Structured Text *)
(* Network 1 *)
ControlloFCUP := NOT S_RC_FineCorsaAlto;
END_TRANSITION

TRANSITION SbloccoUp:
_LD_ (* Ladder Diagram *)
NETWORK 1
	[S_RC_FineCorsaAlto]
_END_LD_
(* the same logic as Structured Text *)
(* Network 1 *)
SbloccoUp := S_RC_FineCorsaAlto;
END_TRANSITION

TRANSITION SbloccoSx:
_LD_ (* Ladder Diagram *)
NETWORK 1
	[/S_RC_FineCorsaSinistra]
_END_LD_
(* the same logic as Structured Text *)
(* Network 1 *)
SbloccoSx := NOT S_RC_FineCorsaSinistra;
END_TRANSITION

TRANSITION TEspelli:
_LD_ (* Ladder Diagram *)
NETWORK 1
	[/Tempo] - [EspelliOK] - [/L7]
_END_LD_
(* the same logic as Structured Text *)
(* Network 1 *)
TEspelli := NOT Tempo AND EspelliOK AND NOT L7;
END_TRANSITION

TRANSITION PresenzaBase:
_LD_ (* Ladder Diagram *)
NETWORK 1
	[AGiostra_Pistone] - T18:TON(IN: *, PT: T#1000ms)
_END_LD_
(* the same logic as Structured Text *)
(* Network 1 *)
T18(IN := AGiostra_Pistone, PT := T#1000ms);
PresenzaBase := T18.Q;
END_TRANSITION

TRANSITION Trans79:
_LD_ (* Ladder Diagram *)
NETWORK 1
	[/AGiostra_Pistone] - [/SGiostra_Presenza] - T19:TON(IN: *, PT: T#1000ms)
_END_LD_
(* the same logic as Structured Text *)
(* Network 1 *)
T19(IN := NOT AGiostra_Pistone AND NOT SGiostra_Presenza, PT := T#1000ms);
Trans79 := T19.Q;
END_TRANSITION

TRANSITION Check+G:
_LD_ (* Ladder Diagram *)
NETWORK 1
	[/L0] - [/L1] - [/L2] - [/L3] - [/L4] - [/L5] - [/L6] - [/GiostraOK] - [/Tempo]
_END_LD_
(* the same logic as Structured Text *)
(* Network 1 *)
Check_G := NOT L0 AND NOT L1 AND NOT L2 AND NOT L3 AND NOT L4 AND NOT L5 AND NOT L6 AND NOT GiostraOK AND NOT Tempo;
END_TRANSITION
END_PROGRAM
